ABB RAPID module: ProgSide2.mod

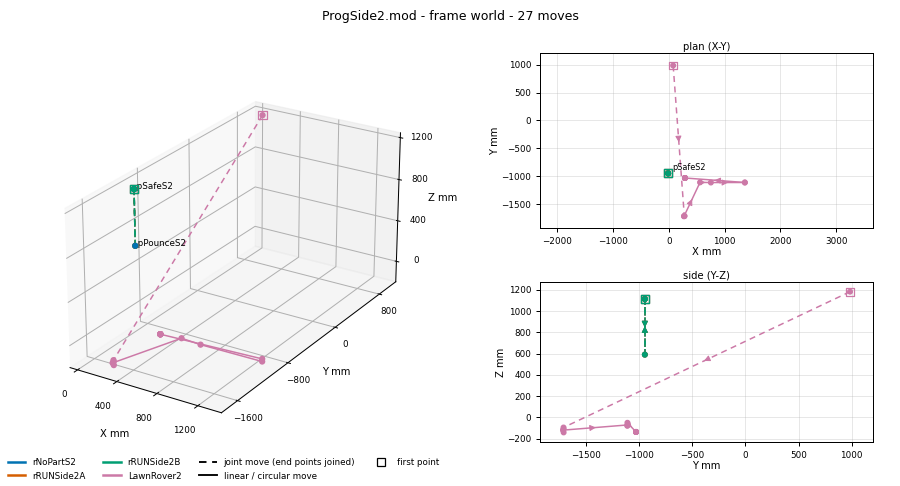
[picture p0: tool path of ProgSide2.mod in frame world, 27 of 27 moves have a stored position in this frame; points joined in program order, loops and branches not executed]
MODULE ProgSide2

	CONST robtarget pPounceOS2:=[[-323.15,704.15,593.73],[0.00135369,-0.9998,0.0053704,-0.0191968],[0,0,-1,0],[9E+09,9E+09,9E+09,9E+09,9E+09,9E+09]];

	PERS welddata weld1:=[10.5833,13.3943,[1,0,25,275.167,0,0,0,0,0],[4,0,23.7,148.167,0,0,0,0,0]];
	PERS welddata weld2:=[12.7,0,[1,0,50,116.417,0,0,0,0,0],[4,0,0,0,0,0,0,0,0]];
	CONST robtarget pPounceS22:=[[375.82,1315.38,357.98],[0.00736884,0.478741,0.877924,0.00116754],[1,-1,1,0],[9E+09,9E+09,9E+09,9E+09,9E+09,9E+09]];
	CONST robtarget pPounceS32:=[[375.82,1315.38,357.98],[0.00736888,0.478742,0.877924,0.00116757],[1,-1,1,0],[9E+09,9E+09,9E+09,9E+09,9E+09,9E+09]];
	CONST robtarget pPounceS42:=[[364.30,-61.64,358.22],[0.0080881,0.475787,0.879523,-0.000148235],[1,-1,1,0],[9E+09,9E+09,9E+09,9E+09,9E+09,9E+09]];
	CONST robtarget pPounceS52:=[[417.56,1241.71,609.54],[0.0379886,-0.00417054,-0.999269,0.00136057],[-2,-1,0,0],[9E+09,9E+09,9E+09,9E+09,9E+09,9E+09]];
	CONST robtarget pPounceS62:=[[417.57,1241.71,609.54],[0.0379873,-0.00416944,-0.999269,0.00136087],[-2,-1,0,0],[9E+09,9E+09,9E+09,9E+09,9E+09,9E+09]];
	CONST robtarget pPounceS72:=[[-13.05,-947.27,590.98],[0.0492186,0.71087,0.699728,-0.0512129],[-2,-1,0,0],[9E+09,9E+09,9E+09,9E+09,9E+09,9E+09]];
	CONST robtarget pPounceS82:=[[420.38,840.44,764.19],[0.0259185,0.406788,0.911848,-0.0488304],[-2,-1,0,0],[9E+09,9E+09,9E+09,9E+09,9E+09,9E+09]];
	PERS welddata weld3:=[12.7,0,[1,0,30,116.417,0,0,0,0,0],[4,0,0,0,0,0,0,0,0]];
	PERS welddata weld4:=[8.46667,13.3943,[1,0,50,78.3167,0,0,0,0,0],[4,0,23.7,148.167,0,0,0,0,0]];
	TASK PERS weavedata weave1:=[1,1,3.81,5.08,5.08,0,0,0,0,0,0,0,0,0,0];
	PERS welddata weld5:=[10.5833,13.3943,[1,0,25,232.833,0,0,0,0,0],[4,0,23.7,148.167,0,0,0,0,0]];
	TASK PERS weavedata weave2:=[1,1,3.81,10.16,1.524,0,0,0,0,0,0,0,0,0,0];
	LOCAL CONST string chassis:="";
!XXXXXXXXXXXXXXXXXXXXXXXXXXXXXXXXXXXXXXXXXXXXXXXXXXXXXXXXXXXXXXXX
!XXXXXXXXXXXXXXXXXXXXXXXXXXXXXXXXXXXXXXXXXXXXXXXXXXXXXXXXXXXXXXXX
!XXXXXXXXXXXXXXXXXXXXXXXXXXXXXXXXXXXXXXXXXXXXXXXXXXXXXXXXXXXXXXXX


!XXXXXXXXXXXXXXXXXXXXXXXXXXXXXXXXXXXXXXXXXXXXXXXXXXXXXXXXXXXXXXXX

     PROC rNoPartS2()
		MoveJ pSafeS2, v800, fine, tWeldGun;
		MoveJ pPounceS2, v800, fine, tWeldGun;
		MoveJ pSafeS2, v800, fine, tWeldGun;
	ENDPROC
!XXXXXXXXXXXXXXXXXXXXXXXXXXXXXXXXXXXXXXXXXXXXXXXXXXXXXXXXXXXXXXXX

!xxxxxxxxxxxxxxxxxxxxxxxxxxxxxxxxxxxxxxxxxxxxxxxxxxxxxxxxxxxxxxx
	PROC rTstA2()
		TPWrite "A S2";
	ENDPROC
	PROC rTstB2()
		TPWrite "B S2";
	ENDPROC
	PROC rRUNSide2A()
		TPWrite "200 Gallon Legs S2 A";
		MoveJ pSafeS2, v800, fine, tWeldGun;
		MoveJ pPounceS2, v800, fine, tWeldGun;
		!Code Goes Here
		MoveJ pSafeS2, v800, fine, tWeldGun;
	ENDPROC
	PROC rRUNSide2B()
		TPWrite "200 Gallon H Frame S2 A";
		MoveJ pSafeS2, v800, fine, tWeldGun;
		MoveJ pPounceS2, v800, fine, tWeldGun;
		!CodeGoes Here
		MoveJ pSafeS2, v800, z10, tWeldGun;
	ENDPROC
	PROC LawnRover2()
		! Chassis
		MoveJ [[76.83,984.99,1183.45],[0.059858,-0.673428,0.735394,0.0459108],[0,-1,0,0],[9E+09,9E+09,9E+09,9E+09,9E+09,9E+09]], v50, z15, tWeldGun;
		MoveJ [[276.91,-1712.92,-95.19],[0.142509,0.476378,0.742146,0.449415],[-2,-2,1,1],[9E+09,9E+09,9E+09,9E+09,9E+09,9E+09]], v50, z15, tWeldGun;
		ArcLStart [[277.91,-1711.84,-108.98],[0.142517,0.476333,0.742133,0.449483],[-2,-2,1,1],[9E+09,9E+09,9E+09,9E+09,9E+09,9E+09]], v5, seam13, weld13, fine, tWeldGun;
		ArcLEnd [[277.91,-1711.84,-141.58],[0.142519,0.476335,0.742132,0.449482],[-2,-2,1,1],[9E+09,9E+09,9E+09,9E+09,9E+09,9E+09]], v5, seam13, weld13, fine, tWeldGun;
		MoveL [[270.94,-1718.17,-120.05],[0.142503,0.476347,0.742161,0.449427],[-2,-2,1,1],[9E+09,9E+09,9E+09,9E+09,9E+09,9E+09]], v50, z50, tWeldGun;
		MoveL [[558.41,-1109.27,-71.06],[0.124309,0.507577,0.785967,0.330408],[-1,-1,0,1],[9E+09,9E+09,9E+09,9E+09,9E+09,9E+09]], v50, z15, tWeldGun;
		ArcLStart [[752.57,-1112.23,-79.31],[0.125463,0.507611,0.786407,0.328868],[-1,-1,0,1],[9E+09,9E+09,9E+09,9E+09,9E+09,9E+09]], v20, seam13, weld13\Weave:=weave1, fine, tWeldGun;
		ArcLEnd [[1361.73,-1111.52,-74.83],[0.124328,0.50762,0.78593,0.330423],[-1,-1,0,1],[9E+09,9E+09,9E+09,9E+09,9E+09,9E+09]], v20, seam13, weld13\Weave:=weave1, fine, tWeldGun;
		MoveL [[1361.67,-1111.46,-50.46],[0.12428,0.507584,0.78597,0.3304],[-1,-1,0,1],[9E+09,9E+09,9E+09,9E+09,9E+09,9E+09]], v50, z15, tWeldGun;
		MoveL [[288.07,-1030.53,-136.86],[0.142555,0.476282,0.742216,0.449388],[-2,-2,0,1],[9E+09,9E+09,9E+09,9E+09,9E+09,9E+09]], v50, z15, tWeldGun;
		ArcLStart [[288.07,-1030.53,-136.86],[0.142555,0.476282,0.742216,0.449389],[-2,-2,0,1],[9E+09,9E+09,9E+09,9E+09,9E+09,9E+09]], v5, seam13, weld13, fine, tWeldGun;
		ArcLEnd [[288.07,-1030.53,-136.86],[0.142554,0.476281,0.742217,0.449389],[-2,-2,0,1],[9E+09,9E+09,9E+09,9E+09,9E+09,9E+09]], v5, seam13, weld13, fine, tWeldGun;
		MoveL [[288.07,-1030.54,-136.86],[0.142555,0.476282,0.742216,0.449388],[-2,-2,0,1],[9E+09,9E+09,9E+09,9E+09,9E+09,9E+09]], v50, z15, tWeldGun;
		MoveL [[288.07,-1030.53,-136.86],[0.142555,0.476282,0.742216,0.449388],[-2,-2,0,1],[9E+09,9E+09,9E+09,9E+09,9E+09,9E+09]], v50, z15, tWeldGun;
		ArcLStart [[288.07,-1030.53,-136.86],[0.142554,0.476282,0.742215,0.44939],[-2,-2,0,1],[9E+09,9E+09,9E+09,9E+09,9E+09,9E+09]], v5, seam13, weld13, fine, tWeldGun;
		ArcLEnd [[288.07,-1030.53,-136.86],[0.142554,0.476281,0.742217,0.449389],[-2,-2,0,1],[9E+09,9E+09,9E+09,9E+09,9E+09,9E+09]], v5, seam13, weld13, fine, tWeldGun;
		MoveL [[288.07,-1030.53,-136.86],[0.142555,0.476283,0.742214,0.44939],[-2,-2,0,1],[9E+09,9E+09,9E+09,9E+09,9E+09,9E+09]], v50, z15, tWeldGun;
		MoveL [[288.07,-1030.53,-136.86],[0.142555,0.476282,0.742216,0.449388],[-2,-2,0,1],[9E+09,9E+09,9E+09,9E+09,9E+09,9E+09]], v50, z15, tWeldGun;
	ENDPROC
ENDMODULE
